(* CODESYS project 04_MySQL_DB_External.ecp

Project tree, tasks and I/O mapping:
  PFC_MySQL_DB_External : 750-8212 PFC200 G2 2ETH RS, WAGO, order no. 0750-8212, version 5.16.3.46
    application Application
      libraries: WagoAppTime, 1.7.3.4 (WAGO); VisuDialogs, * (System); WagoAppSQL_MySQL, 1.6.1.1 (WAGO)
      task PLC_Task (cyclic, interval t#30ms, priority 13) calls PLC_PRG
      task Task_SQL (cyclic, interval 50 ms, priority 15) calls PRG_SQL
      program PLC_PRG [ST]
      program PRG_SQL [FBD]
      FBs/
        function block FbSQLInsertCommand_dbTraining [ST]
      data type typByte2String
      data type typState
    ProjectConfiguration
    Kbus : Kbus, WAGO, version 1.4.0.2
        unmapped channels: K-BUS diagnostics
    MODBUS
      MODBUS : MODBUS, WAGO, order no. n/a, version 1.1.1.16
    Serial
      COM1 : COM1, WAGO, version 0.0.0.19
    Common.PCI
    EtherNet/IP
      Ethernet : Ethernet, WAGO, version 35.16.0.0
          settings: IPAddress = [192, 168, 1, 212]; SubnetMask = [0, 0, 0, 0]; MACAddress = [16#00, 16#00, 16#00, 16#00, 16#00, 16#00]; NetworkInterfaceName = 'br0'; NetworkInterfaceName = "br0"
  libraries: VisuSymbols, 3.5.17.0 (System); WagoVisuIcons, 1.1.0.4 (WAGO)
  text list GlobalTextList
  00000000-0000-0000-0000-000000000000|C:\Users\u0100068\AppData\Local\Temp\1a00fa59f6a2463e8b93f081f6ce7d9f\e868b832187f4f1a859da50215710801\Project.xml
*)

// PFC_MySQL_DB_External/Application/typByte2String
TYPE typByte2String :
UNION		// convert an array of byte to a readable string
	sData:	STRING(MYSQL_MAX_ROW_SIZE);
	abData:	ARRAY [0..MYSQL_MAX_ROW_SIZE] OF BYTE;
END_UNION
END_TYPE

// PFC_MySQL_DB_External/Application/typState
{attribute 'qualified_only'}
{attribute 'strict'}
TYPE typState :
(
	eIdle,
	eHandleLogin,
	eProcessSqlExecute,
	eHandleLogout,
	eErrorHandling
);
END_TYPE

// PFC_MySQL_DB_External/Application/PLC_PRG
PROGRAM PLC_PRG
VAR
	timDelay			: TON;
	dtLocalTime			: DATE_AND_TIME;
	sTime				: STRING(8);
	sDate				: STRING(10);

	xRandomActive		: BOOL := TRUE;
	rOffsetTemperature	: REAL;
	rOffsetVoltage		: REAL;
	xDigitalInput8		: BOOL;

	rTemperatureStatic	: REAL := 23.5;
	rVoltageStatic		: REAL := 5.834;
	rTemperature		: REAL;
	rVoltage			: REAL;
END_VAR

// get date and time of the controller only every second, because it's stressy
timDelay(IN := NOT timDelay.Q, PT := T#1S);
IF timDelay.Q THEN
	dtLocalTime	:= FuGetLocalDateAndTime();
	sTime		:= WagoAppString.FuTodToString(bFormat := 1, todInput := TO_TOD(dtLocalTime));
	sDate		:= WagoAppString.FuDateToString(bFormat := 0, datInput := TO_DATE(dtLocalTime));

	// generate some data to fill database
	IF xRandomActive THEN
		// create some randomness for temperature value
		rOffsetTemperature	:= 8.34 * SIN(TO_REAL(PRG_SQL.a) / 30.0);
		// create some randomness for voltage value
		rOffsetVoltage		:= 3.78 * SIN(TO_REAL(PRG_SQL.a) / 12.8);
	ELSE
		rOffsetVoltage		:= 0;
		rOffsetTemperature	:= 0;
	END_IF
	
	// toggle input
	xDigitalInput8			:= NOT xDigitalInput8;
END_IF;

// add some changes
rTemperature	:= rTemperatureStatic 	+ rOffsetTemperature;
rVoltage		:= rVoltageStatic		+ rOffsetVoltage;

END_PROGRAM

// PFC_MySQL_DB_External/Application/PRG_SQL
PROGRAM PRG_SQL
VAR
	sIP_LinuxDB			: STRING := '192.168.1.212';
	sUserLinuxDB		: STRING := 'dozent';
	sPwdLinuxDB			: STRING := 'Master!';
	sDatabaseName		: STRING := 'dbTraining';
	sTableName			: STRING := 'TblTraining';

//_______________________________________________________________

	oFBdbTraining_Format9: FbSQLInsertCommand_dbTraining;
	xConnect			: BOOL;
	sDate				: STRING := 'Date';
	sTime				: STRING := 'Time';
	sTemp				: STRING := 'Temperature';
	sDigitalInput		: STRING := 'EmergencyStop';
	sVoltage			: STRING := 'Voltage';
	xTriggerWrite		: BOOL;
	xConnectedToLinuxDatabase: BOOL;

	FbMySqlQuery		: FbMySql_Query;
	aSqlCommand			: ARRAY [0..MYSQL_SQL_UPPER_BOUND] OF STRING(MYSQL_SQL_LENGTH)
						:= ['SELECT * FROM dbTraining.TblTraining WHERE EmergencyStop =  1 AND Date > $272020-01-20$27 LIMIT 10', 10('')];
	xTriggerQuery		: BOOL;
	typResultSqlQuery	: typMySql_ResultSet;
	xBusyQuery			: BOOL;
	xErrorQuery			: BOOL;
	oStatusQuery		: WagoSysErrorBase.FbResult;
	sStatusQuery		: STRING(200);

	a:INT;
	
END_VAR

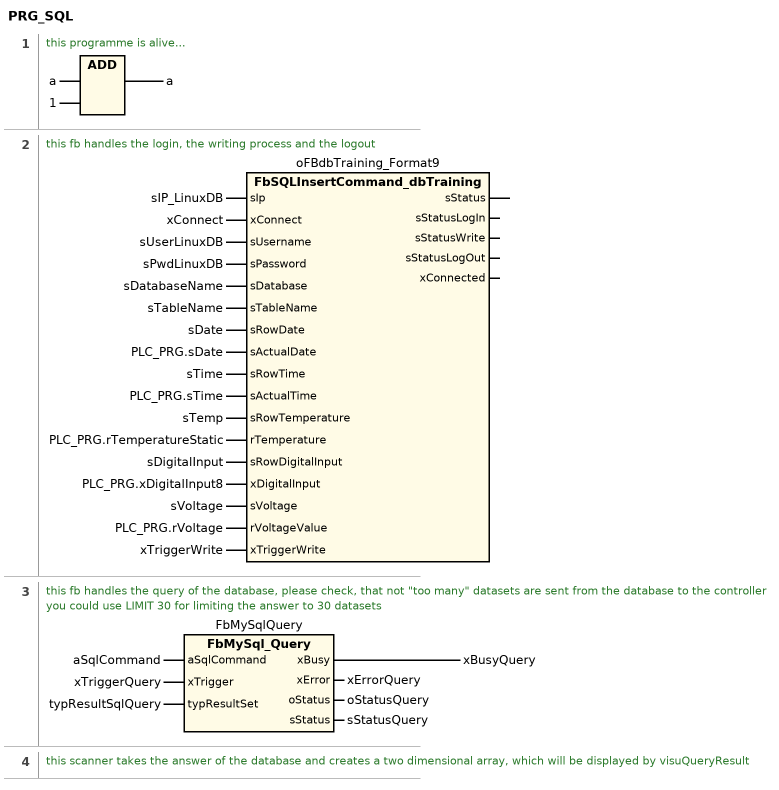
// NETWORK 1
// this programme is alive...
a := a + 1;

// NETWORK 2
// this fb handles the login, the writing process and the logout
oFBdbTraining_Format9(
    sIp := sIP_LinuxDB,
    xConnect := xConnect,
    sUsername := sUserLinuxDB,
    sPassword := sPwdLinuxDB,
    sDatabase := sDatabaseName,
    sTableName := sTableName,
    sRowDate := sDate,
    sActualDate := PLC_PRG.sDate,
    sRowTime := sTime,
    sActualTime := PLC_PRG.sTime,
    sRowTemperature := sTemp,
    rTemperature := PLC_PRG.rTemperatureStatic,
    sRowDigitalInput := sDigitalInput,
    xDigitalInput := PLC_PRG.xDigitalInput8,
    sVoltage := sVoltage,
    rVoltageValue := PLC_PRG.rVoltage,
    xTriggerWrite := xTriggerWrite); // FbSQLInsertCommand_dbTraining

// NETWORK 3
// this fb handles the query of the database, please check, that not "too many" datasets are sent from the database to the controller
// you could use LIMIT 30 for limiting the answer to 30 datasets
FbMySqlQuery(
    aSqlCommand := aSqlCommand,
    xTrigger := xTriggerQuery,
    typResultSet := typResultSqlQuery,
    xError => xErrorQuery,
    oStatus => oStatusQuery,
    sStatus => sStatusQuery); // FbMySql_Query
xBusyQuery := FbMySqlQuery.xBusy;

// NETWORK 4
// this scanner takes the answer of the database and creates a two dimensional array, which will be displayed by visuQueryResult

END_PROGRAM

// PFC_MySQL_DB_External/Application/FBs/FbSQLInsertCommand_dbTraining
FUNCTION_BLOCK FbSQLInsertCommand_dbTraining
VAR_INPUT
	sIp					: STRING := '192.168.1.2';				// ip address of the server
	xConnect			: BOOL;					// connect to the data base
	sUsername			: STRING;				// database username
	sPassword			: STRING;				// database password
	sDatabase			: STRING;				// database name which you want to acccess
	sTableName			: STRING;				// table which belongs to your chosen database 
	
	sRowDate			: STRING;				// first row of your table
	sActualDate			: STRING(10);
	
	sRowTime			: STRING;				// second row of your table
	sActualTime			: STRING(8);
	
	sRowTemperature		: STRING;				// third row of your table
	rTemperature		: REAL;
	
	sRowDigitalInput	: STRING;				// fourth row of your table
	xDigitalInput		: BOOL;
	
	sVoltage			: STRING;				// fifth row of your table
	rVoltageValue		: REAL;
END_VAR
VAR_OUTPUT
	sStatus				: STRING;
	sStatusLogIn		: STRING(200);
	sStatusWrite		: STRING(200);
	sStatusLogOut		: STRING(200);
	xConnected			: BOOL;
END_VAR
VAR_IN_OUT
	xTriggerWrite		: BOOL;
END_VAR
VAR
	xInit				: BOOL := TRUE;
	aSqlCommand			: ARRAY [0..MYSQL_SQL_UPPER_BOUND] OF STRING(MYSQL_SQL_LENGTH);
	sActualDigitalInput	: STRING(20);

	iState				: INT;
	FbSqlLogin		: FbMySql_Login;
	xTriggerLogin		: BOOL;
	xBusyLogIn			: BOOL;
	xErrorLogIn			: BOOL;
	
	fbSqlExecute01		: FbMySql_Execute;
	
	xBusyWrite			: BOOL;
	xErrorWrite			: BOOL;
	
	fbSqlLogout01		: FbMySql_Logout;
	xTriggerLogout		: BOOL;
	xBusyLogOut			: BOOL;
	xErrorLogOut		: BOOL;
END_VAR

// initialisation procedure
IF xInit THEN
	aSqlCommand[0] := Format6(
		sFormat	:= 'INSERT INTO %s(%s,%s,%s,%s,%s) ',
		p1		:= ADR(sTableName),
		p2		:= ADR(sRowDate),
		p3		:= ADR(sRowTime),
		p4		:= ADR(sRowTemperature),
		p5		:= ADR(sRowDigitalInput),
		p6		:= ADR(sVoltage));
	xInit := FALSE;			// initialisation process is over
END_IF

//---------------------------------------------------------------------------------------------------------------------------------------------------------------------------------------------------------------------------------------
// since Format5 uses pointers it is necessary to use variables after typecasting- otherwise an error will occur
sActualDigitalInput	:= TO_STRING(xDigitalInput);

aSqlCommand[1] := Format5(
	sFormat	:= 'VALUES($27%s$27,$27%s$27,%4.1f,%s,%5.2f)',		// $27 ==> ' ==> inverted comma
	p1		:= ADR(sActualDate),
	p2		:= ADR(sActualTime),
	p3		:= ADR(rTemperature),
	p4		:= ADR(sActualDigitalInput),
	p5		:= ADR(rVoltageValue));

// target: INSERT INTO 'dbTraining'('Date','Time','Temperature',EmergencyStop,'Voltage') VALUES('2017-10-31',10:33:05,23.3,true,8.7)

// ATTENTION: The function block Login01 has to be called within every PLC cycle!!!
FbSqlLogin(
	sHost		:= sIp,
	//uiPort	:= ,
	sUsername	:= sUsername,
	sPassword	:= sPassword,
	sDatabase	:= sDatabase,
	xTrigger	:= xTriggerLogin,
	xBusy		=> xBusyLogIn,
	xError		=> xErrorLogIn,
	//oStatus	=> ,
	sStatus		=> sStatusLogIn,
	xConnected	=> xConnected);

CASE iState OF
//------------------------------------------------------------------------------------------
	typState.eIdle:
		sStatus := 'SQL idle';
		IF xConnect THEN
			xTriggerLogin := TRUE;
			iState := typState.eHandleLogin;
		END_IF

//------------------------------------------------------------------------------------------
	typState.eHandleLogin:
		IF NOT xTriggerLogin THEN
			IF xConnected THEN
				iState	:= typState.eProcessSqlExecute;
				sStatus	:= 'SQL connected';
			ELSE
				iState	:= typState.eErrorHandling;
				sStatus	:= 'SQL connect error';
			END_IF
		END_IF
//------------------------------------------------------------------------------------------	
	typState.eProcessSqlExecute:
		fbSqlExecute01(
			aSqlCommand	:= aSqlCommand,
			xTrigger	:= xTriggerWrite,
			xBusy		=> xBusyWrite,
			xError		=> xErrorWrite,
			//oStatus	=> ,
			sStatus		=> sStatusWrite);
		IF NOT xConnect THEN
			xTriggerLogout := TRUE;
			iState := typState.eHandleLogout;
		END_IF

//------------------------------------------------------------------------------------------	
	typState.eHandleLogout:
		fbSqlLogout01(
			xTrigger	:= xTriggerLogout,
			xBusy		=> xBusyLogOut,
			xError		=> xErrorLogOut,
			//oStatus	=> ,
			sStatus		=> sStatusLogOut);
		IF NOT xTriggerLogout THEN
			IF NOT xErrorLogOut THEN
				iState	:= typState.eIdle;
				sStatus	:= 'SQL disconnected';
			ELSE
				iState	:= typState.eErrorHandling;
				sStatus	:= 'SQL Logout Error';
			END_IF;
		END_IF;
	typState.eErrorHandling:
		sStatus := 'Error Handling tbd';

END_CASE
//------------------------------------------------------------------------------------------

END_FUNCTION_BLOCK
